TYPE ST_HW_OutputsProfileCheck :
STRUCT

END_STRUCT
END_TYPE

(* stored: Version 1.1.0.1, ProductVersion 3.1.4024.9
   DUT ST_HW_OutputsProfileCheck: Id {c41013a4-1983-4ec7-9d08-e42a12753647} *)
